{attribute 'qualified_only'}
{attribute 'strict'}
{attribute 'to_string'}
TYPE Axis_e :
(
    ST110_01Y,  //  0
    ST110_02Z,  //  1
    ST110_03Z,  //  2
    ST110_04Z,  //  3
	ST110_10W,  //  4
    ST115_01Y,  //  5
    ST115_02Z,  //  6
    ST115_03Z,  //  7
    ST115_04Z,  //  8
	ST115_10W,  //  9
    ST120_01Y,  // 10
    ST120_02Z,  // 11
    ST125_01Y,  // 12
    ST125_02Z,  // 13
	ST125_10W,  // 14
	ST130_01Z,  // 15
	ST130_10Z,  // 16
	ST135_01Z,  // 17
	ST135_10Z,  // 18
	ST145_01Y,  // 19
	ST145_02Z,  // 20
	ST145_10W,  // 21
	ST160_01Z,  // 22
	ST165_01Z,  // 23
	ST170_01Z,  // 24
	ST180_01Y,  // 25
	ST180_02Z,  // 26
	ST180_10Z,  // 27
	ST185_01Y,  // 28
	ST185_02Z,  // 29
	ST185_10Z,  // 30
    _max
);
END_TYPE

(* stored: Version 1.1.0.1, ProductVersion 3.1.4024.6
   EnumerationTextList Axis_e: Id {c595cd03-c145-453e-b0fc-824a9ab61cfe} *)
